ABB RobotStudio station: gripper.rsstn

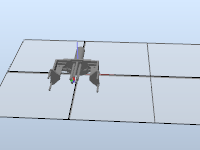
Station gripper (saved by RobotStudio 21.2.9526.0)
Layout (positions relative to the parent item):
  - GripperRueda [mechanism, from Gripper\GripperRueda.rslib] at (0, 0, 0) mm; joint values [0, 0, 0] (rad or m)
